PROGRAM MAIN
VAR
	i1,i2:INT;
	i3:INT:=5;
END_VAR
//An UPS is necessary to save the persistent Data, if it's not available other options are also possible, such as:
//Save to retain data / text files/Databases or simple use the FB_WritePersistentData and soon as a new error occur to make sure it's gonna be persistent
//Note : leaving Checks activated on a running machine can have negative effects on the performance
//As you find out what's the problem you should also remove checks from your code

//Here we call the program which handles the diagnosis
//
prgDiag();

i1:=i2/i3;

END_PROGRAM

(* stored: Version 1.1.0.1, ProductVersion 3.1.4024.9
   POU MAIN: Id {3ad06a0b-d0de-4cb6-a41a-d10b92c01dcc}, SpecialFunc None *)
